TYPE ST_CompensationDiagnostic :
STRUCT
    bError : BOOL;                          // Hata durumu
    eError : E_CompensationError;           // Hata kodu
    wsErrorMessage : WSTRING(255);          // Hata mesajı
END_STRUCT
END_TYPE

(* stored: Version 1.1.0.1, ProductVersion 3.1.4024.15
   DUT ST_CompensationDiagnostic: Id {7c5ba760-7796-460f-81b8-052cad4e039c} *)
